PROGRAM PistonOnly
VAR_IN_OUT
	smc : AirPiston;
END_VAR
VAR
	ready : BOOL;
	in : BOOL;
	out : BOOL;
END_VAR

smc.bEnable := TRUE;

smc();

IF NOT ready THEN
	ready := smc.homingSequence();
	RETURN;
END_IF


//IF NOT (in OR out) THEN
	//smc.stop();
//END_IF

IF in THEN
	smc.extend();
	out := FALSE;
END_IF

IF out THEN
	smc.retract();
	in := FALSE;
END_IF

IF smc.innerLimit THEN
	in := FALSE;
END_IF

IF smc.home THEN
	out := FALSE;
END_IF

END_PROGRAM

(* stored: Version 1.1.0.1, ProductVersion 3.1.4024.11
   POU PistonOnly: Id {d6a96585-c3b9-4bd2-bcab-43977d1dfb12}, SpecialFunc None *)
